KUKA KRL data list: 1p_mit_komp.dat

&ACCESS RVP
&REL 14
&PARAM DISKPATH = KRC:\R1\Program\SprutCam\GRUNDEISTELLUNGEN ROBOTER
DEFDAT  mit_komp
;FOLD EXTERNAL DECLARATIONS;%{PE}%MKUKATPBASIS,%CEXT,%VCOMMON,%P
;FOLD BASISTECH EXT;%{PE}%MKUKATPBASIS,%CEXT,%VEXT,%P
EXT  BAS (BAS_COMMAND  :IN,REAL  :IN )
DECL INT SUCCESS
;ENDFOLD (BASISTECH EXT)
;FOLD USER EXT;%{E}%MKUKATPUSER,%CEXT,%VEXT,%P
;Make your modifications here

;ENDFOLD (USER EXT)
;ENDFOLD (EXTERNAL DECLARATIONS)
DECL BASIS_SUGG_T LAST_BASIS={POINT1[] "P15                     ",POINT2[] "P15                     ",CP_PARAMS[] "CPDAT0                  ",PTP_PARAMS[] "PDAT15                  ",CONT[] "                        ",CP_VEL[] "2.0                     ",PTP_VEL[] "30                      ",SYNC_PARAMS[] "SYNCDAT                 ",SPL_NAME[] "S0                      ",A_PARAMS[] "ADAT0                   "}

DECL E6POS XP1={X 1590.08093,Y -19.7581234,Z 524.630554,A 159.345505,B 86.6105499,C 111.772629,S 22,T 50,E1 0.00497351913,E2 20160.0,E3 0.0,E4 0.0,E5 0.0,E6 0.0}
DECL FDAT FP1={TOOL_NO 12,BASE_NO 0,IPO_FRAME #BASE,POINT2[] " ",TQ_STATE FALSE}
DECL PDAT PPDAT1={VEL 100.000,ACC 50.0000,APO_DIST 100.000,APO_MODE #CDIS,GEAR_JERK 50.0000,EXAX_IGN 0}

ENDDAT
